{attribute 'qualified_only'}
{attribute 'strict'}
{attribute 'to_string'}
TYPE E_CilinderZuignap :
(
	Ingetrokken,
	Verlengt,
	Error
);
END_TYPE

(* stored: Version 1.1.0.1
   DUT E_CilinderZuignap: Id {0d8a10dc-bd12-44ef-844e-2edf3ec2cd1c} *)
